// TIA Portal V16 export
// export: Created 2024-09-05T17:40:13.8974602Z, ExportSetting WithDefaults, DisplayName Totally Integrated Automation Portal, DisplayVersion V16 Update 6, DisplayName TIA Portal Version Control Interface, DisplayVersion V16 Update 2, DisplayName TIA Portal Openness, DisplayVersion V16 Update 6, DisplayName STEP 7 Professional, DisplayVersion V16 Update 6, DisplayName STEP 7 Safety, DisplayVersion V16, DisplayName WinCC Advanced, DisplayVersion V16 Update 6
TYPE "UDT_Digiforce"
// stored: IsFailsafeCompliant false
   STRUCT
      programActual : USInt;
      programOK : Bool;
      ProgramChangeNOK : Bool;
      programSet : USInt;
      ActualWay : Real;
      ActualForce : Real;
      Ready : Bool;
      ResultOK : Bool;
      ResultNOK : Bool;
      Auto : Bool;
      Start : Bool;
      Running : Bool;
      TareX : Bool;
   END_STRUCT;
END_TYPE
